LIN {X 0,Y 241.571,Z 805.243,A -85,B 0,C 180,E1 1203.684,E2 1203.684} C_VEL
LIN {X 0,Y 247.431,Z 809.251,A -85,B 0,C 180,E1 1199.707,E2 1199.707} C_VEL
LIN {X 0,Y 250.618,Z 811.939,A -85,B 0,C 180,E1 1197.052,E2 1197.052} C_VEL
LIN {X 0,Y 255.628,Z 815.815,A -85,B 0,C 180,E1 1192.538,E2 1192.538} C_VEL
LIN {X 0,Y 260.599,Z 818.711,A -85,B 0,C 180,E1 1187.958,E2 1187.958} C_VEL
LIN {X 0,Y 261.974,Z 819.683,A -85,B 0,C 180,E1 1186.177,E2 1186.177} C_VEL
LIN {X 0,Y 264.278,Z 822.142,A -85,B 0,C 180,E1 1181.788,E2 1181.788} C_VEL
LIN {X 0,Y 265.852,Z 823.476,A -85,B 0,C 180,E1 1178.216,E2 1178.216} C_VEL
LIN {X 0,Y 266.855,Z 824.18,A -85,B 0,C 180,E1 1175.159,E2 1175.159} C_VEL
LIN {X 0,Y 267.405,Z 824.567,A -85,B 0,C 180,E1 1171.928,E2 1171.928} C_VEL
LIN {X 0,Y 267.503,Z 824.602,A -85,B 0,C 180,E1 1168.501,E2 1168.501} C_VEL
LIN {X 0,Y 266.809,Z 824.172,A -85,B 0,C 180,E1 1164.624,E2 1164.624} C_VEL
LIN {X 0,Y 265.597,Z 823.259,A -85,B 0,C 180,E1 1161.121,E2 1161.121} C_VEL
LIN {X 0,Y 263.851,Z 821.702,A -85,B 0,C 180,E1 1157.304,E2 1157.304} C_VEL
LIN {X 0,Y 261.509,Z 819.124,A -85,B 0,C 180,E1 1152.982,E2 1152.982} C_VEL
LIN {X 0,Y 258.841,Z 817.772,A -85,B 0,C 180,E1 1150.452,E2 1150.452} C_VEL
LIN {X 0,Y 256.402,Z 817.327,A -85,B 0,C 180,E1 1148.951,E2 1148.951} C_VEL
LIN {X 0,Y 250.102,Z 817.193,A -85,B 0,C 180,E1 1146.411,E2 1146.411} C_VEL
LIN {X 0,Y 245.371,Z 816.618,A -85,B 0,C 180,E1 1144.345,E2 1144.345} C_VEL
LIN {X 0,Y 243.571,Z 815.677,A -85,B 0,C 180,E1 1143.12,E2 1143.12} C_VEL
LIN {X 0,Y 240.616,Z 813.189,A -85,B 0,C 180,E1 1140.638,E2 1140.638} C_VEL
LIN {X 0,Y 234.191,Z 808.745,A -85,B 0,C 180,E1 1136.289,E2 1136.289} C_VEL
LIN {X 0,Y 228.396,Z 804.049,A -85,B 0,C 180,E1 1132.384,E2 1132.384} C_VEL
LIN {X 0,Y 218.07,Z 796.351,A -85,B 0,C 180,E1 1126.021,E2 1126.021} C_VEL
LIN {X 0,Y 208.768,Z 790.269,A -85,B 0,C 180,E1 1119.927,E2 1119.927} C_VEL
LIN {X 0,Y 193.411,Z 803.184,A -85,B 0,C 180,E1 1122.334,E2 1122.334} C_VEL
LIN {X 0,Y 177.615,Z 814.532,A -85,B 0,C 180,E1 1125.28,E2 1125.28} C_VEL
LIN {X 0,Y 161.491,Z 824.391,A -85,B 0,C 180,E1 1128.984,E2 1128.984} C_VEL
LIN {X 0,Y 145.341,Z 832.727,A -85,B 0,C 180,E1 1133.729,E2 1133.729} C_VEL
LIN {X 0,Y 130.379,Z 839.113,A -85,B 0,C 180,E1 1139.594,E2 1139.594} C_VEL
LIN {X 0,Y 116.492,Z 844.004,A -85,B 0,C 180,E1 1147.28,E2 1147.28} C_VEL
LIN {X 0,Y 105.301,Z 847.033,A -85,B 0,C 180,E1 1156.828,E2 1156.828} C_VEL
LIN {X 0,Y 98.168,Z 848.251,A -85,B 0,C 180,E1 1167.665,E2 1167.665} C_VEL
LIN {X 0,Y 97.266,Z 848.365,A -85,B 0,C 180,E1 1170,E2 1170} C_VEL
LIN {X 0,Y 104.158,Z 847.276,A -85,B 0,C 180,E1 1181.86,E2 1181.86} C_VEL
LIN {X 0,Y 115.295,Z 844.363,A -85,B 0,C 180,E1 1191.894,E2 1191.894} C_VEL
LIN {X 0,Y 128.965,Z 839.667,A -85,B 0,C 180,E1 1199.747,E2 1199.747} C_VEL
LIN {X 0,Y 143.784,Z 833.459,A -85,B 0,C 180,E1 1205.74,E2 1205.74} C_VEL
LIN {X 0,Y 159.832,Z 825.327,A -85,B 0,C 180,E1 1210.585,E2 1210.585} C_VEL
LIN {X 0,Y 175.89,Z 815.636,A -85,B 0,C 180,E1 1214.361,E2 1214.361} C_VEL
LIN {X 0,Y 192.523,Z 803.858,A -85,B 0,C 180,E1 1217.514,E2 1217.514} C_VEL
LIN {X 0,Y 207.75,Z 791.179,A -85,B 0,C 180,E1 1219.926,E2 1219.926} C_VEL
LIN {X 0,Y 208.906,Z 790.205,A -85,B 0,C 180,E1 1220.06,E2 1220.06} C_VEL
LIN {X 0,Y 219.341,Z 797.322,A -85,B 0,C 180,E1 1213.137,E2 1213.137} C_VEL
LIN {X 0,Y 229.518,Z 804.819,A -85,B 0,C 180,E1 1206.953,E2 1206.953} C_VEL
LIN {X 0,Y 235.927,Z 810.04,A -85,B 0,C 180,E1 1202.529,E2 1202.529} C_VEL
LIN {X 0,Y 241.591,Z 813.831,A -85,B 0,C 180,E1 1198.69,E2 1198.69} C_VEL
LIN {X 0,Y 246.575,Z 818.132,A -85,B 0,C 180,E1 1194.176,E2 1194.176} C_VEL
LIN {X 0,Y 251.386,Z 821.277,A -85,B 0,C 180,E1 1189.759,E2 1189.759} C_VEL
LIN {X 0,Y 254.404,Z 822.806,A -85,B 0,C 180,E1 1186.907,E2 1186.907} C_VEL
LIN {X 0,Y 256.658,Z 825.293,A -85,B 0,C 180,E1 1182.829,E2 1182.829} C_VEL
LIN {X 0,Y 258.465,Z 826.898,A -85,B 0,C 180,E1 1178.901,E2 1178.901} C_VEL
LIN {X 0,Y 259.61,Z 827.709,A -85,B 0,C 180,E1 1175.525,E2 1175.525} C_VEL
LIN {X 0,Y 260.237,Z 828.148,A -85,B 0,C 180,E1 1172.202,E2 1172.202} C_VEL
LIN {X 0,Y 260.358,Z 828.214,A -85,B 0,C 180,E1 1169.12,E2 1169.12} C_VEL
LIN {X 0,Y 259.817,Z 827.9,A -85,B 0,C 180,E1 1165.144,E2 1165.144} C_VEL
LIN {X 0,Y 258.455,Z 826.885,A -85,B 0,C 180,E1 1161.098,E2 1161.098} C_VEL
LIN {X 0,Y 256.865,Z 825.487,A -85,B 0,C 180,E1 1157.631,E2 1157.631} C_VEL
LIN {X 0,Y 254.588,Z 823.004,A -85,B 0,C 180,E1 1153.34,E2 1153.34} C_VEL
LIN {X 0,Y 251.095,Z 821.118,A -85,B 0,C 180,E1 1149.969,E2 1149.969} C_VEL
LIN {X 0,Y 246.557,Z 818.126,A -85,B 0,C 180,E1 1145.811,E2 1145.811} C_VEL
LIN {X 0,Y 243.571,Z 815.677,A -85,B 0,C 180,E1 1143.12,E2 1143.12} C_VEL
LIN {X 0,Y 241.186,Z 814.652,A -85,B 0,C 180,E1 1141.677,E2 1141.677} C_VEL
LIN {X 0,Y 235.768,Z 813.842,A -85,B 0,C 180,E1 1139.652,E2 1139.652} C_VEL
LIN {X 0,Y 227.805,Z 812.371,A -85,B 0,C 180,E1 1136.778,E2 1136.778} C_VEL
LIN {X 0,Y 225.724,Z 811.177,A -85,B 0,C 180,E1 1135.642,E2 1135.642} C_VEL
LIN {X 0,Y 221.245,Z 807.582,A -85,B 0,C 180,E1 1132.668,E2 1132.668} C_VEL
LIN {X 0,Y 210.893,Z 800.282,A -85,B 0,C 180,E1 1126.086,E2 1126.086} C_VEL
LIN {X 0,Y 205.938,Z 797.244,A -85,B 0,C 180,E1 1122.887,E2 1122.887} C_VEL
LIN {X 0,Y 190.335,Z 809.479,A -85,B 0,C 180,E1 1125.681,E2 1125.681} C_VEL
LIN {X 0,Y 175.132,Z 819.746,A -85,B 0,C 180,E1 1128.964,E2 1128.964} C_VEL
LIN {X 0,Y 158.983,Z 828.979,A -85,B 0,C 180,E1 1133.313,E2 1133.313} C_VEL
LIN {X 0,Y 144.292,Z 836.035,A -85,B 0,C 180,E1 1138.425,E2 1138.425} C_VEL
LIN {X 0,Y 129.595,Z 841.892,A -85,B 0,C 180,E1 1145.379,E2 1145.379} C_VEL
LIN {X 0,Y 117.064,Z 845.841,A -85,B 0,C 180,E1 1154.139,E2 1154.139} C_VEL
LIN {X 0,Y 108.029,Z 847.814,A -85,B 0,C 180,E1 1164.69,E2 1164.69} C_VEL
LIN {X 0,Y 105.426,Z 848.124,A -85,B 0,C 180,E1 1170,E2 1170} C_VEL
LIN {X 0,Y 112.034,Z 847.075,A -85,B 0,C 180,E1 1180.802,E2 1180.802} C_VEL
LIN {X 0,Y 122.392,Z 844.297,A -85,B 0,C 180,E1 1190.066,E2 1190.066} C_VEL
LIN {X 0,Y 135.485,Z 839.7,A -85,B 0,C 180,E1 1197.705,E2 1197.705} C_VEL
LIN {X 0,Y 149.772,Z 833.556,A -85,B 0,C 180,E1 1203.647,E2 1203.647} C_VEL
LIN {X 0,Y 166.14,Z 825.083,A -85,B 0,C 180,E1 1208.746,E2 1208.746} C_VEL
LIN {X 0,Y 181.829,Z 815.391,A -85,B 0,C 180,E1 1212.561,E2 1212.561} C_VEL
LIN {X 0,Y 197.252,Z 804.289,A -85,B 0,C 180,E1 1215.619,E2 1215.619} C_VEL
LIN {X 0,Y 205.946,Z 797.252,A -85,B 0,C 180,E1 1217.106,E2 1217.106} C_VEL
LIN {X 0,Y 212.978,Z 801.72,A -85,B 0,C 180,E1 1212.533,E2 1212.533} C_VEL
LIN {X 0,Y 222.929,Z 808.794,A -85,B 0,C 180,E1 1206.3,E2 1206.3} C_VEL
LIN {X 0,Y 229.468,Z 814.048,A -85,B 0,C 180,E1 1201.818,E2 1201.818} C_VEL
LIN {X 0,Y 234.739,Z 817.563,A -85,B 0,C 180,E1 1198.182,E2 1198.182} C_VEL
LIN {X 0,Y 239.861,Z 821.879,A -85,B 0,C 180,E1 1193.534,E2 1193.534} C_VEL
LIN {X 0,Y 244.44,Z 824.864,A -85,B 0,C 180,E1 1189.348,E2 1189.348} C_VEL
LIN {X 0,Y 247.403,Z 826.429,A -85,B 0,C 180,E1 1186.433,E2 1186.433} C_VEL
LIN {X 0,Y 249.748,Z 828.99,A -85,B 0,C 180,E1 1182.015,E2 1182.015} C_VEL
LIN {X 0,Y 251.389,Z 830.35,A -85,B 0,C 180,E1 1178.232,E2 1178.232} C_VEL
LIN {X 0,Y 252.513,Z 831.153,A -85,B 0,C 180,E1 1174.77,E2 1174.77} C_VEL
LIN {X 0,Y 253.142,Z 831.571,A -85,B 0,C 180,E1 1170.905,E2 1170.905} C_VEL
LIN {X 0,Y 252.872,Z 831.392,A -85,B 0,C 180,E1 1167.054,E2 1167.054} C_VEL
LIN {X 0,Y 252.067,Z 830.824,A -85,B 0,C 180,E1 1163.623,E2 1163.623} C_VEL
LIN {X 0,Y 250.517,Z 829.695,A -85,B 0,C 180,E1 1159.654,E2 1159.654} C_VEL
LIN {X 0,Y 248.572,Z 827.829,A -85,B 0,C 180,E1 1155.732,E2 1155.732} C_VEL
LIN {X 0,Y 246.826,Z 826.071,A -85,B 0,C 180,E1 1152.893,E2 1152.893} C_VEL
LIN {X 0,Y 242.802,Z 823.869,A -85,B 0,C 180,E1 1149.154,E2 1149.154} C_VEL
LIN {X 0,Y 237.804,Z 820.313,A -85,B 0,C 180,E1 1144.605,E2 1144.605} C_VEL
LIN {X 0,Y 233.786,Z 816.896,A -85,B 0,C 180,E1 1141.101,E2 1141.101} C_VEL
LIN {X 0,Y 227.169,Z 812.34,A -85,B 0,C 180,E1 1136.622,E2 1136.622} C_VEL
LIN {X 0,Y 225.724,Z 811.177,A -85,B 0,C 180,E1 1135.642,E2 1135.642} C_VEL
LIN {X 0,Y 222.496,Z 809.65,A -85,B 0,C 180,E1 1134.047,E2 1134.047} C_VEL
LIN {X 0,Y 215.713,Z 808.301,A -85,B 0,C 180,E1 1131.746,E2 1131.746} C_VEL
LIN {X 0,Y 208.332,Z 806.725,A -85,B 0,C 180,E1 1129.074,E2 1129.074} C_VEL
LIN {X 0,Y 206.131,Z 805.617,A -85,B 0,C 180,E1 1127.852,E2 1127.852} C_VEL
LIN {X 0,Y 203.146,Z 803.962,A -85,B 0,C 180,E1 1126.006,E2 1126.006} C_VEL
LIN {X 0,Y 187.103,Z 815.704,A -85,B 0,C 180,E1 1129.312,E2 1129.312} C_VEL
LIN {X 0,Y 171.822,Z 825.277,A -85,B 0,C 180,E1 1133.176,E2 1133.176} C_VEL
LIN {X 0,Y 156.672,Z 833.316,A -85,B 0,C 180,E1 1138.016,E2 1138.016} C_VEL
LIN {X 0,Y 142.812,Z 839.46,A -85,B 0,C 180,E1 1143.828,E2 1143.828} C_VEL
LIN {X 0,Y 130.145,Z 844.051,A -85,B 0,C 180,E1 1151.176,E2 1151.176} C_VEL
LIN {X 0,Y 119.709,Z 846.911,A -85,B 0,C 180,E1 1160.384,E2 1160.384} C_VEL
LIN {X 0,Y 113.592,Z 847.883,A -85,B 0,C 180,E1 1170,E2 1170} C_VEL
LIN {X 0,Y 120.107,Z 846.831,A -85,B 0,C 180,E1 1180.068,E2 1180.068} C_VEL
LIN {X 0,Y 130.145,Z 844.051,A -85,B 0,C 180,E1 1188.824,E2 1188.824} C_VEL
LIN {X 0,Y 142.812,Z 839.46,A -85,B 0,C 180,E1 1196.172,E2 1196.172} C_VEL
LIN {X 0,Y 156.797,Z 833.257,A -85,B 0,C 180,E1 1202.03,E2 1202.03} C_VEL
LIN {X 0,Y 172.606,Z 824.838,A -85,B 0,C 180,E1 1207.044,E2 1207.044} C_VEL
LIN {X 0,Y 187.927,Z 815.152,A -85,B 0,C 180,E1 1210.874,E2 1210.874} C_VEL
LIN {X 0,Y 203.351,Z 803.878,A -85,B 0,C 180,E1 1213.984,E2 1213.984} C_VEL
LIN {X 0,Y 208.882,Z 807.581,A -85,B 0,C 180,E1 1210.255,E2 1210.255} C_VEL
LIN {X 0,Y 216.301,Z 812.586,A -85,B 0,C 180,E1 1205.58,E2 1205.58} C_VEL
LIN {X 0,Y 223.318,Z 818.002,A -85,B 0,C 180,E1 1200.753,E2 1200.753} C_VEL
LIN {X 0,Y 227.829,Z 821.081,A -85,B 0,C 180,E1 1197.594,E2 1197.594} C_VEL
LIN {X 0,Y 232.511,Z 824.921,A -85,B 0,C 180,E1 1193.304,E2 1193.304} C_VEL
LIN {X 0,Y 236.697,Z 827.703,A -85,B 0,C 180,E1 1189.494,E2 1189.494} C_VEL
LIN {X 0,Y 240.105,Z 829.608,A -85,B 0,C 180,E1 1186.2,E2 1186.2} C_VEL
LIN {X 0,Y 242.327,Z 831.94,A -85,B 0,C 180,E1 1181.905,E2 1181.905} C_VEL
LIN {X 0,Y 243.938,Z 833.305,A -85,B 0,C 180,E1 1178.248,E2 1178.248} C_VEL
LIN {X 0,Y 245.176,Z 834.222,A -85,B 0,C 180,E1 1174.444,E2 1174.444} C_VEL
LIN {X 0,Y 245.688,Z 834.566,A -85,B 0,C 180,E1 1170.466,E2 1170.466} C_VEL
LIN {X 0,Y 245.443,Z 834.378,A -85,B 0,C 180,E1 1166.964,E2 1166.964} C_VEL
LIN {X 0,Y 244.565,Z 833.754,A -85,B 0,C 180,E1 1163.427,E2 1163.427} C_VEL
LIN {X 0,Y 242.909,Z 832.512,A -85,B 0,C 180,E1 1159.326,E2 1159.326} C_VEL
LIN {X 0,Y 240.776,Z 830.411,A -85,B 0,C 180,E1 1155.081,E2 1155.081} C_VEL
LIN {X 0,Y 239.384,Z 829.149,A -85,B 0,C 180,E1 1152.986,E2 1152.986} C_VEL
LIN {X 0,Y 234.828,Z 826.562,A -85,B 0,C 180,E1 1148.782,E2 1148.782} C_VEL
LIN {X 0,Y 229.8,Z 822.851,A -85,B 0,C 180,E1 1144.209,E2 1144.209} C_VEL
LIN {X 0,Y 226.539,Z 820.12,A -85,B 0,C 180,E1 1141.409,E2 1141.409} C_VEL
LIN {X 0,Y 219.742,Z 815.384,A -85,B 0,C 180,E1 1136.821,E2 1136.821} C_VEL
LIN {X 0,Y 214.512,Z 811.258,A -85,B 0,C 180,E1 1133.268,E2 1133.268} C_VEL
LIN {X 0,Y 206.131,Z 805.617,A -85,B 0,C 180,E1 1127.852,E2 1127.852} C_VEL
LIN {X 0,Y 205.537,Z 806.099,A -85,B 0,C 180,E1 1127.97,E2 1127.97} C_VEL
LIN {X 0,Y 205.112,Z 808.121,A -85,B 0,C 180,E1 1129.091,E2 1129.091} C_VEL
LIN {X 0,Y 206.966,Z 812.608,A -85,B 0,C 180,E1 1132.341,E2 1132.341} C_VEL
LIN {X 0,Y 212.015,Z 818.017,A -85,B 0,C 180,E1 1136.913,E2 1136.913} C_VEL
LIN {X 0,Y 219.563,Z 823.232,A -85,B 0,C 180,E1 1142.029,E2 1142.029} C_VEL
LIN {X 0,Y 224.132,Z 827.034,A -85,B 0,C 180,E1 1146.099,E2 1146.099} C_VEL
LIN {X 0,Y 228.79,Z 830.212,A -85,B 0,C 180,E1 1150.336,E2 1150.336} C_VEL
LIN {X 0,Y 232.486,Z 832.206,A -85,B 0,C 180,E1 1153.767,E2 1153.767} C_VEL
LIN {X 0,Y 234.677,Z 834.483,A -85,B 0,C 180,E1 1157.95,E2 1157.95} C_VEL
LIN {X 0,Y 236.567,Z 836.139,A -85,B 0,C 180,E1 1162.227,E2 1162.227} C_VEL
LIN {X 0,Y 237.7,Z 836.9,A -85,B 0,C 180,E1 1165.899,E2 1165.899} C_VEL
LIN {X 0,Y 238.099,Z 837.169,A -85,B 0,C 180,E1 1169.278,E2 1169.278} C_VEL
LIN {X 0,Y 237.968,Z 837.078,A -85,B 0,C 180,E1 1172.408,E2 1172.408} C_VEL
LIN {X 0,Y 237.256,Z 836.592,A -85,B 0,C 180,E1 1175.805,E2 1175.805} C_VEL
LIN {X 0,Y 235.742,Z 835.464,A -85,B 0,C 180,E1 1179.767,E2 1179.767} C_VEL
LIN {X 0,Y 233.601,Z 833.432,A -85,B 0,C 180,E1 1184.121,E2 1184.121} C_VEL
LIN {X 0,Y 232.216,Z 832.092,A -85,B 0,C 180,E1 1186.509,E2 1186.509} C_VEL
LIN {X 0,Y 227.177,Z 829.19,A -85,B 0,C 180,E1 1191.155,E2 1191.155} C_VEL
LIN {X 0,Y 221.919,Z 825.207,A -85,B 0,C 180,E1 1195.914,E2 1195.914} C_VEL
LIN {X 0,Y 219.086,Z 822.929,A -85,B 0,C 180,E1 1198.292,E2 1198.292} C_VEL
LIN {X 0,Y 211.878,Z 817.909,A -85,B 0,C 180,E1 1203.188,E2 1203.188} C_VEL
LIN {X 0,Y 207.172,Z 814.425,A -85,B 0,C 180,E1 1206.413,E2 1206.413} C_VEL
LIN {X 0,Y 200.608,Z 810.29,A -85,B 0,C 180,E1 1210.717,E2 1210.717} C_VEL
LIN {X 0,Y 185.419,Z 820.742,A -85,B 0,C 180,E1 1207.152,E2 1207.152} C_VEL
LIN {X 0,Y 170.929,Z 829.301,A -85,B 0,C 180,E1 1202.956,E2 1202.956} C_VEL
LIN {X 0,Y 156.773,Z 836.402,A -85,B 0,C 180,E1 1197.747,E2 1197.747} C_VEL
LIN {X 0,Y 143.526,Z 841.862,A -85,B 0,C 180,E1 1191.238,E2 1191.238} C_VEL
LIN {X 0,Y 132.482,Z 845.481,A -85,B 0,C 180,E1 1183.53,E2 1183.53} C_VEL
LIN {X 0,Y 124.056,Z 847.369,A -85,B 0,C 180,E1 1174.16,E2 1174.16} C_VEL
LIN {X 0,Y 121.763,Z 847.641,A -85,B 0,C 180,E1 1170,E2 1170} C_VEL
LIN {X 0,Y 128.201,Z 846.587,A -85,B 0,C 180,E1 1160.574,E2 1160.574} C_VEL
LIN {X 0,Y 137.952,Z 843.806,A -85,B 0,C 180,E1 1152.278,E2 1152.278} C_VEL
LIN {X 0,Y 150.231,Z 839.219,A -85,B 0,C 180,E1 1145.211,E2 1145.211} C_VEL
LIN {X 0,Y 163.69,Z 833.076,A -85,B 0,C 180,E1 1139.538,E2 1139.538} C_VEL
LIN {X 0,Y 178.447,Z 825.032,A -85,B 0,C 180,E1 1134.753,E2 1134.753} C_VEL
LIN {X 0,Y 193.374,Z 815.463,A -85,B 0,C 180,E1 1130.891,E2 1130.891} C_VEL
LIN {X 0,Y 200.659,Z 810.328,A -85,B 0,C 180,E1 1129.321,E2 1129.321} C_VEL
LIN {X 0,Y 209.081,Z 815.695,A -85,B 0,C 180,E1 1134.833,E2 1134.833} C_VEL
LIN {X 0,Y 212.015,Z 818.017,A -85,B 0,C 180,E1 1136.913,E2 1136.913} C_VEL
LIN {X 0,Y 213.631,Z 820.009,A -85,B 0,C 180,E1 1138.575,E2 1138.575} C_VEL
LIN {X 0,Y 214.34,Z 823.486,A -85,B 0,C 180,E1 1141.11,E2 1141.11} C_VEL
LIN {X 0,Y 215.162,Z 828.031,A -85,B 0,C 180,E1 1144.841,E2 1144.841} C_VEL
LIN {X 0,Y 216.13,Z 829.13,A -85,B 0,C 180,E1 1145.976,E2 1145.976} C_VEL
LIN {X 0,Y 221.042,Z 832.532,A -85,B 0,C 180,E1 1150.444,E2 1150.444} C_VEL
LIN {X 0,Y 224.871,Z 834.577,A -85,B 0,C 180,E1 1153.998,E2 1153.998} C_VEL
LIN {X 0,Y 227.161,Z 836.959,A -85,B 0,C 180,E1 1158.319,E2 1158.319} C_VEL
LIN {X 0,Y 228.966,Z 838.471,A -85,B 0,C 180,E1 1162.473,E2 1162.473} C_VEL
LIN {X 0,Y 230.085,Z 839.176,A -85,B 0,C 180,E1 1166.263,E2 1166.263} C_VEL
LIN {X 0,Y 230.415,Z 839.426,A -85,B 0,C 180,E1 1169.751,E2 1169.751} C_VEL
LIN {X 0,Y 230.227,Z 839.258,A -85,B 0,C 180,E1 1173.022,E2 1173.022} C_VEL
LIN {X 0,Y 229.164,Z 838.631,A -85,B 0,C 180,E1 1177.017,E2 1177.017} C_VEL
LIN {X 0,Y 227.394,Z 837.168,A -85,B 0,C 180,E1 1181.155,E2 1181.155} C_VEL
LIN {X 0,Y 225.34,Z 835.062,A -85,B 0,C 180,E1 1185.176,E2 1185.176} C_VEL
LIN {X 0,Y 223.97,Z 834.169,A -85,B 0,C 180,E1 1186.868,E2 1186.868} C_VEL
LIN {X 0,Y 219.36,Z 831.448,A -85,B 0,C 180,E1 1191.105,E2 1191.105} C_VEL
LIN {X 0,Y 214.217,Z 827.528,A -85,B 0,C 180,E1 1195.768,E2 1195.768} C_VEL
LIN {X 0,Y 211.562,Z 825.463,A -85,B 0,C 180,E1 1197.932,E2 1197.932} C_VEL
LIN {X 0,Y 203.595,Z 819.998,A -85,B 0,C 180,E1 1203.426,E2 1203.426} C_VEL
LIN {X 0,Y 199.519,Z 817.339,A -85,B 0,C 180,E1 1206.24,E2 1206.24} C_VEL
LIN {X 0,Y 197.917,Z 816.532,A -85,B 0,C 180,E1 1207.18,E2 1207.18} C_VEL
LIN {X 0,Y 183.71,Z 825.666,A -85,B 0,C 180,E1 1203.345,E2 1203.345} C_VEL
LIN {X 0,Y 169.442,Z 833.504,A -85,B 0,C 180,E1 1198.552,E2 1198.552} C_VEL
LIN {X 0,Y 156.505,Z 839.526,A -85,B 0,C 180,E1 1192.936,E2 1192.936} C_VEL
LIN {X 0,Y 144.284,Z 844.098,A -85,B 0,C 180,E1 1185.679,E2 1185.679} C_VEL
LIN {X 0,Y 135.099,Z 846.604,A -85,B 0,C 180,E1 1177.549,E2 1177.549} C_VEL
LIN {X 0,Y 129.941,Z 847.4,A -85,B 0,C 180,E1 1170,E2 1170} C_VEL
LIN {X 0,Y 136.31,Z 846.342,A -85,B 0,C 180,E1 1161.139,E2 1161.139} C_VEL
LIN {X 0,Y 145.805,Z 843.56,A -85,B 0,C 180,E1 1153.261,E2 1153.261} C_VEL
LIN {X 0,Y 157.729,Z 838.979,A -85,B 0,C 180,E1 1146.462,E2 1146.462} C_VEL
LIN {X 0,Y 170.815,Z 832.835,A -85,B 0,C 180,E1 1140.934,E2 1140.934} C_VEL
LIN {X 0,Y 185.197,Z 824.788,A -85,B 0,C 180,E1 1136.216,E2 1136.216} C_VEL
LIN {X 0,Y 198.101,Z 816.527,A -85,B 0,C 180,E1 1132.862,E2 1132.862} C_VEL
LIN {X 0,Y 202.46,Z 819.184,A -85,B 0,C 180,E1 1135.738,E2 1135.738} C_VEL
LIN {X 0,Y 210.574,Z 824.818,A -85,B 0,C 180,E1 1141.421,E2 1141.421} C_VEL
LIN {X 0,Y 213.52,Z 826.941,A -85,B 0,C 180,E1 1143.586,E2 1143.586} C_VEL
LIN {X 0,Y 216.13,Z 829.13,A -85,B 0,C 180,E1 1145.976,E2 1145.976} C_VEL
LIN {X 0,Y 217.447,Z 830.995,A -85,B 0,C 180,E1 1147.935,E2 1147.935} C_VEL
LIN {X 0,Y 217.498,Z 833.736,A -85,B 0,C 180,E1 1150.789,E2 1150.789} C_VEL
LIN {X 0,Y 217.529,Z 836.966,A -85,B 0,C 180,E1 1154.729,E2 1154.729} C_VEL
LIN {X 0,Y 217.729,Z 837.251,A -85,B 0,C 180,E1 1155.166,E2 1155.166} C_VEL
LIN {X 0,Y 219.913,Z 839.379,A -85,B 0,C 180,E1 1159.522,E2 1159.522} C_VEL
LIN {X 0,Y 221.453,Z 840.528,A -85,B 0,C 180,E1 1163.259,E2 1163.259} C_VEL
LIN {X 0,Y 222.428,Z 841.178,A -85,B 0,C 180,E1 1166.908,E2 1166.908} C_VEL
LIN {X 0,Y 222.712,Z 841.37,A -85,B 0,C 180,E1 1170.772,E2 1170.772} C_VEL
LIN {X 0,Y 222.1,Z 840.989,A -85,B 0,C 180,E1 1174.648,E2 1174.648} C_VEL
LIN {X 0,Y 220.759,Z 840.01,A -85,B 0,C 180,E1 1178.596,E2 1178.596} C_VEL
LIN {X 0,Y 218.868,Z 838.389,A -85,B 0,C 180,E1 1182.666,E2 1182.666} C_VEL
LIN {X 0,Y 216.856,Z 836.533,A -85,B 0,C 180,E1 1186.059,E2 1186.059} C_VEL
LIN {X 0,Y 211.698,Z 833.52,A -85,B 0,C 180,E1 1190.79,E2 1190.79} C_VEL
LIN {X 0,Y 206.734,Z 829.754,A -85,B 0,C 180,E1 1195.292,E2 1195.292} C_VEL
LIN {X 0,Y 204.123,Z 827.799,A -85,B 0,C 180,E1 1197.415,E2 1197.415} C_VEL
LIN {X 0,Y 195.612,Z 822.321,A -85,B 0,C 180,E1 1203.442,E2 1203.442} C_VEL
LIN {X 0,Y 182.119,Z 830.352,A -85,B 0,C 180,E1 1199.249,E2 1199.249} C_VEL
LIN {X 0,Y 168.141,Z 837.428,A -85,B 0,C 180,E1 1193.731,E2 1193.731} C_VEL
LIN {X 0,Y 156.267,Z 842.418,A -85,B 0,C 180,E1 1187.501,E2 1187.501} C_VEL
LIN {X 0,Y 145.989,Z 845.741,A -85,B 0,C 180,E1 1179.859,E2 1179.859} C_VEL
LIN {X 0,Y 139.315,Z 847.011,A -85,B 0,C 180,E1 1172.056,E2 1172.056} C_VEL
LIN {X 0,Y 138.124,Z 847.158,A -85,B 0,C 180,E1 1170,E2 1170} C_VEL
LIN {X 0,Y 144.478,Z 846.088,A -85,B 0,C 180,E1 1161.594,E2 1161.594} C_VEL
LIN {X 0,Y 153.858,Z 843.257,A -85,B 0,C 180,E1 1154.037,E2 1154.037} C_VEL
LIN {X 0,Y 165.553,Z 838.618,A -85,B 0,C 180,E1 1147.475,E2 1147.475} C_VEL
LIN {X 0,Y 178.704,Z 832.258,A -85,B 0,C 180,E1 1141.968,E2 1141.968} C_VEL
LIN {X 0,Y 193.516,Z 823.665,A -85,B 0,C 180,E1 1137.146,E2 1137.146} C_VEL
LIN {X 0,Y 195.694,Z 822.386,A -85,B 0,C 180,E1 1136.625,E2 1136.625} C_VEL
LIN {X 0,Y 204.707,Z 828.142,A -85,B 0,C 180,E1 1142.985,E2 1142.985} C_VEL
LIN {X 0,Y 209.535,Z 832.009,A -85,B 0,C 180,E1 1147.263,E2 1147.263} C_VEL
LIN {X 0,Y 214.185,Z 835.094,A -85,B 0,C 180,E1 1151.493,E2 1151.493} C_VEL
LIN {X 0,Y 217.53,Z 837.007,A -85,B 0,C 180,E1 1154.792,E2 1154.792} C_VEL
LIN {X 0,Y 217.729,Z 837.251,A -85,B 0,C 180,E1 1155.166,E2 1155.166} C_VEL
LIN {X 0,Y 217.847,Z 838.498,A -85,B 0,C 180,E1 1157.031,E2 1157.031} C_VEL
LIN {X 0,Y 215.999,Z 840.367,A -85,B 0,C 180,E1 1159.903,E2 1159.903} C_VEL
LIN {X 0,Y 213.965,Z 842.087,A -85,B 0,C 180,E1 1163.306,E2 1163.306} C_VEL
LIN {X 0,Y 214.02,Z 842.451,A -85,B 0,C 180,E1 1164.512,E2 1164.512} C_VEL
LIN {X 0,Y 214.798,Z 842.935,A -85,B 0,C 180,E1 1168.4,E2 1168.4} C_VEL
LIN {X 0,Y 214.732,Z 842.909,A -85,B 0,C 180,E1 1171.868,E2 1171.868} C_VEL
LIN {X 0,Y 214.05,Z 842.427,A -85,B 0,C 180,E1 1175.36,E2 1175.36} C_VEL
LIN {X 0,Y 212.611,Z 841.397,A -85,B 0,C 180,E1 1179.2,E2 1179.2} C_VEL
LIN {X 0,Y 210.405,Z 839.416,A -85,B 0,C 180,E1 1183.745,E2 1183.745} C_VEL
LIN {X 0,Y 209.007,Z 838.221,A -85,B 0,C 180,E1 1185.823,E2 1185.823} C_VEL
LIN {X 0,Y 203.68,Z 835.084,A -85,B 0,C 180,E1 1190.698,E2 1190.698} C_VEL
LIN {X 0,Y 197.763,Z 830.551,A -85,B 0,C 180,E1 1196.094,E2 1196.094} C_VEL
LIN {X 0,Y 192.996,Z 828.023,A -85,B 0,C 180,E1 1199.281,E2 1199.281} C_VEL
LIN {X 0,Y 179.567,Z 835.343,A -85,B 0,C 180,E1 1194.333,E2 1194.333} C_VEL
LIN {X 0,Y 167.835,Z 840.668,A -85,B 0,C 180,E1 1188.765,E2 1188.765} C_VEL
LIN {X 0,Y 156.995,Z 844.615,A -85,B 0,C 180,E1 1181.759,E2 1181.759} C_VEL
LIN {X 0,Y 149.194,Z 846.576,A -85,B 0,C 180,E1 1174.228,E2 1174.228} C_VEL
LIN {X 0,Y 146.31,Z 846.916,A -85,B 0,C 180,E1 1170,E2 1170} C_VEL
LIN {X 0,Y 152.564,Z 845.854,A -85,B 0,C 180,E1 1162.09,E2 1162.09} C_VEL
LIN {X 0,Y 161.62,Z 843.07,A -85,B 0,C 180,E1 1154.94,E2 1154.94} C_VEL
LIN {X 0,Y 172.917,Z 838.496,A -85,B 0,C 180,E1 1148.637,E2 1148.637} C_VEL
LIN {X 0,Y 185.328,Z 832.355,A -85,B 0,C 180,E1 1143.399,E2 1143.399} C_VEL
LIN {X 0,Y 193.13,Z 827.971,A -85,B 0,C 180,E1 1140.698,E2 1140.698} C_VEL
LIN {X 0,Y 198.346,Z 831.031,A -85,B 0,C 180,E1 1144.429,E2 1144.429} C_VEL
LIN {X 0,Y 204.345,Z 835.515,A -85,B 0,C 180,E1 1149.913,E2 1149.913} C_VEL
LIN {X 0,Y 209.338,Z 838.393,A -85,B 0,C 180,E1 1154.487,E2 1154.487} C_VEL
LIN {X 0,Y 211.718,Z 840.654,A -85,B 0,C 180,E1 1158.836,E2 1158.836} C_VEL
LIN {X 0,Y 213.391,Z 841.988,A -85,B 0,C 180,E1 1162.732,E2 1162.732} C_VEL
LIN {X 0,Y 214.02,Z 842.451,A -85,B 0,C 180,E1 1164.512,E2 1164.512} C_VEL
LIN {X 0,Y 213.73,Z 842.928,A -85,B 0,C 180,E1 1166.284,E2 1166.284} C_VEL
LIN {X 0,Y 211.436,Z 843.523,A -85,B 0,C 180,E1 1168.762,E2 1168.762} C_VEL
LIN {X 0,Y 206.968,Z 843.981,A -85,B 0,C 180,E1 1172.964,E2 1172.964} C_VEL
LIN {X 0,Y 206.477,Z 843.902,A -85,B 0,C 180,E1 1174.062,E2 1174.062} C_VEL
LIN {X 0,Y 205.01,Z 842.872,A -85,B 0,C 180,E1 1178.413,E2 1178.413} C_VEL
LIN {X 0,Y 202.912,Z 841.017,A -85,B 0,C 180,E1 1182.811,E2 1182.811} C_VEL
LIN {X 0,Y 201.419,Z 839.72,A -85,B 0,C 180,E1 1185.253,E2 1185.253} C_VEL
LIN {X 0,Y 196.486,Z 836.85,A -85,B 0,C 180,E1 1189.759,E2 1189.759} C_VEL
LIN {X 0,Y 190.984,Z 833.026,A -85,B 0,C 180,E1 1194.841,E2 1194.841} C_VEL
LIN {X 0,Y 178.904,Z 839.047,A -85,B 0,C 180,E1 1189.592,E2 1189.592} C_VEL
LIN {X 0,Y 168.163,Z 843.362,A -85,B 0,C 180,E1 1183.408,E2 1183.408} C_VEL
LIN {X 0,Y 159.644,Z 845.851,A -85,B 0,C 180,E1 1176.473,E2 1176.473} C_VEL
LIN {X 0,Y 154.5,Z 846.674,A -85,B 0,C 180,E1 1170,E2 1170} C_VEL
LIN {X 0,Y 160.706,Z 845.609,A -85,B 0,C 180,E1 1162.493,E2 1162.493} C_VEL
LIN {X 0,Y 169.573,Z 842.824,A -85,B 0,C 180,E1 1155.662,E2 1155.662} C_VEL
LIN {X 0,Y 180.592,Z 838.253,A -85,B 0,C 180,E1 1149.587,E2 1149.587} C_VEL
LIN {X 0,Y 191.008,Z 833.05,A -85,B 0,C 180,E1 1145.187,E2 1145.187} C_VEL
LIN {X 0,Y 196.645,Z 836.96,A -85,B 0,C 180,E1 1150.393,E2 1150.393} C_VEL
LIN {X 0,Y 201.876,Z 839.993,A -85,B 0,C 180,E1 1155.18,E2 1155.18} C_VEL
LIN {X 0,Y 204.169,Z 842.185,A -85,B 0,C 180,E1 1159.754,E2 1159.754} C_VEL
LIN {X 0,Y 205.764,Z 843.413,A -85,B 0,C 180,E1 1163.583,E2 1163.583} C_VEL
LIN {X 0,Y 206.763,Z 844.09,A -85,B 0,C 180,E1 1167.506,E2 1167.506} C_VEL
LIN {X 0,Y 206.882,Z 844.174,A -85,B 0,C 180,E1 1171.385,E2 1171.385} C_VEL
LIN {X 0,Y 206.477,Z 843.902,A -85,B 0,C 180,E1 1174.062,E2 1174.062} C_VEL
LIN {X 0,Y 205.207,Z 843.715,A -85,B 0,C 180,E1 1175.874,E2 1175.874} C_VEL
LIN {X 0,Y 201.585,Z 843.286,A -85,B 0,C 180,E1 1178.343,E2 1178.343} C_VEL
LIN {X 0,Y 195.598,Z 842.102,A -85,B 0,C 180,E1 1182.231,E2 1182.231} C_VEL
LIN {X 0,Y 194.433,Z 841.393,A -85,B 0,C 180,E1 1183.68,E2 1183.68} C_VEL
LIN {X 0,Y 193.048,Z 840.523,A -85,B 0,C 180,E1 1185.316,E2 1185.316} C_VEL
LIN {X 0,Y 188.311,Z 838.011,A -85,B 0,C 180,E1 1189.542,E2 1189.542} C_VEL
LIN {X 0,Y 178.018,Z 842.399,A -85,B 0,C 180,E1 1183.976,E2 1183.976} C_VEL
LIN {X 0,Y 169.215,Z 845.285,A -85,B 0,C 180,E1 1177.469,E2 1177.469} C_VEL
LIN {X 0,Y 162.92,Z 846.408,A -85,B 0,C 180,E1 1170.352,E2 1170.352} C_VEL
LIN {X 0,Y 162.925,Z 846.407,A -85,B 0,C 180,E1 1169.642,E2 1169.642} C_VEL
LIN {X 0,Y 169.215,Z 845.285,A -85,B 0,C 180,E1 1162.531,E2 1162.531} C_VEL
LIN {X 0,Y 178.018,Z 842.399,A -85,B 0,C 180,E1 1156.024,E2 1156.024} C_VEL
LIN {X 0,Y 188.456,Z 838.006,A -85,B 0,C 180,E1 1150.474,E2 1150.474} C_VEL
LIN {X 0,Y 194.108,Z 841.08,A -85,B 0,C 180,E1 1155.686,E2 1155.686} C_VEL
LIN {X 0,Y 196.423,Z 843.246,A -85,B 0,C 180,E1 1160.33,E2 1160.33} C_VEL
LIN {X 0,Y 198.103,Z 844.511,A -85,B 0,C 180,E1 1164.497,E2 1164.497} C_VEL
LIN {X 0,Y 198.943,Z 844.997,A -85,B 0,C 180,E1 1168.56,E2 1168.56} C_VEL
LIN {X 0,Y 198.824,Z 844.922,A -85,B 0,C 180,E1 1172.306,E2 1172.306} C_VEL
LIN {X 0,Y 197.893,Z 844.328,A -85,B 0,C 180,E1 1176.091,E2 1176.091} C_VEL
LIN {X 0,Y 196.281,Z 843.108,A -85,B 0,C 180,E1 1179.973,E2 1179.973} C_VEL
LIN {X 0,Y 194.433,Z 841.393,A -85,B 0,C 180,E1 1183.68,E2 1183.68} C_VEL
LIN {X 0,Y 193.21,Z 841.382,A -85,B 0,C 180,E1 1183.896,E2 1183.896} C_VEL
LIN {X 0,Y 190.174,Z 841.785,A -85,B 0,C 180,E1 1183.611,E2 1183.611} C_VEL
LIN {X 0,Y 185.976,Z 842.682,A -85,B 0,C 180,E1 1182.446,E2 1182.446} C_VEL
LIN {X 0,Y 179.08,Z 844.624,A -85,B 0,C 180,E1 1178.421,E2 1178.421} C_VEL
LIN {X 0,Y 174.645,Z 845.694,A -85,B 0,C 180,E1 1174.557,E2 1174.557} C_VEL
LIN {X 0,Y 170.92,Z 846.188,A -85,B 0,C 180,E1 1169.955,E2 1169.955} C_VEL
LIN {X 0,Y 177.248,Z 845.067,A -85,B 0,C 180,E1 1162.979,E2 1162.979} C_VEL
LIN {X 0,Y 186.005,Z 842.154,A -85,B 0,C 180,E1 1156.636,E2 1156.636} C_VEL
LIN {X 0,Y 186.439,Z 842.027,A -85,B 0,C 180,E1 1156.451,E2 1156.451} C_VEL
LIN {X 0,Y 188.472,Z 843.784,A -85,B 0,C 180,E1 1160.555,E2 1160.555} C_VEL
LIN {X 0,Y 190.099,Z 844.94,A -85,B 0,C 180,E1 1164.568,E2 1164.568} C_VEL
LIN {X 0,Y 190.906,Z 845.451,A -85,B 0,C 180,E1 1168.199,E2 1168.199} C_VEL
LIN {X 0,Y 190.884,Z 845.451,A -85,B 0,C 180,E1 1171.801,E2 1171.801} C_VEL
LIN {X 0,Y 190.098,Z 844.94,A -85,B 0,C 180,E1 1175.432,E2 1175.432} C_VEL
LIN {X 0,Y 188.47,Z 843.785,A -85,B 0,C 180,E1 1179.443,E2 1179.443} C_VEL
LIN {X 0,Y 186.396,Z 842.002,A -85,B 0,C 180,E1 1183.601,E2 1183.601} C_VEL
LIN {X 0,Y 177.727,Z 844.96,A -85,B 0,C 180,E1 1177.434,E2 1177.434} C_VEL
LIN {X 0,Y 174.645,Z 845.694,A -85,B 0,C 180,E1 1174.557,E2 1174.557} C_VEL
LIN {X 0,Y 174.222,Z 845.94,A -85,B 0,C 180,E1 1173.126,E2 1173.126} C_VEL
LIN {X 0,Y 175.985,Z 846.017,A -85,B 0,C 180,E1 1171.01,E2 1171.01} C_VEL
LIN {X 0,Y 180.926,Z 845.722,A -85,B 0,C 180,E1 1167.608,E2 1167.608} C_VEL
LIN {X 0,Y 181.406,Z 845.672,A -85,B 0,C 180,E1 1167.139,E2 1167.139} C_VEL
LIN {X 0,Y 182.484,Z 845.539,A -85,B 0,C 180,E1 1166,E2 1166} C_VEL
LIN {X 0,Y 182.974,Z 845.815,A -85,B 0,C 180,E1 1169.687,E2 1169.687} C_VEL
LIN {X 0,Y 182.555,Z 845.568,A -85,B 0,C 180,E1 1173.768,E2 1173.768} C_VEL
LIN {X 0,Y 182.483,Z 845.539,A -85,B 0,C 180,E1 1173.999,E2 1173.999} C_VEL
LIN {X 0,Y 179.089,Z 845.947,A -85,B 0,C 180,E1 1170,E2 1170} C_VEL
LIN {X 0,Y 181.406,Z 845.672,A -85,B 0,C 180,E1 1167.139,E2 1167.139} C_VEL
LIN {X 0,Y 181.986,Z 847.671,A -85,B 0,C 180,E1 1166.515,E2 1166.515} C_VEL
LIN {X 0,Y 181.986,Z 875,A -85,B 0,C 180,E1 1166.515,E2 1166.515} C_VEL
LIN {X 0,Y 181.986,Z 875,A -85,B 0,C 180,E1 1166.515,E2 1166.515}

QRS_NEXT_CUT()

QRS_NEXT()
QRS_HOME()

END
